// TIA Portal V19 export
FUNCTION "webserver" : Void   // FC1, LAD
   VAR_TEMP
      RET_VAL_1 : Int;
   END_VAR
BEGIN

REGION Network 1
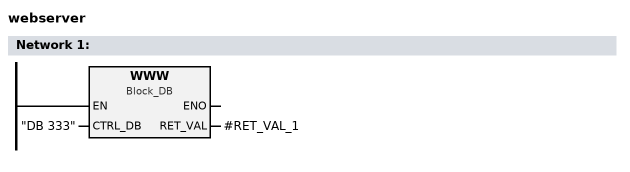
   RUNG wire#powerrail
      { S7_Templates := "value_type := Block_DB" } WWW(CTRL_DB := "DB 333", RET_VAL => #RET_VAL_1)
   END_RUNG
   // the same network as SCL:
   #RET_VAL_1 := WWW(CTRL_DB := "DB 333");
END_REGION
END_FUNCTION
